// TwinCAT 3 PLC project MAS418_Crane_Simulator_1
// ProgramVersion: 3.1.4024.0
// libraries:
//   Tc2_Standard, * (Beckhoff Automation GmbH)
//   Tc2_System, * (Beckhoff Automation GmbH)
//   Tc3_Module, * (Beckhoff Automation GmbH)
// project tree:
//   Crane_Controller/Enums/ E_ControlBoxSwitchMode.TcDUT, E_RunningStates.TcDUT
//   Crane_Controller/GVL/ G_HMI.TcGVL
//   Crane_Controller/Interfaces/ I_CraneControlBox.TcIO
//   Crane_Controller/POU/ FB_AutoMode.TcPOU, FB_ClosedLoopControl.TcPOU, FB_ControlBox.TcPOU, FB_ManualMode.TcPOU, FB_MotionReferenceGenerator.TcPOU, FB_OpenLoopControl.TcPOU, FB_RealControlBox.TcPOU, FB_VirtualControlBox.TcPOU
//   Crane_Controller/Structs/ ST_CraneHMIData.TcDUT, ST_MotionGeneratorData.TcDUT, ST_OpenLoopControlData.TcDUT
//   / GlobalTextList.TcGTLO, PlcTask.TcTTO, Simulator_1.TcTTO, Visualization Manager.TcVMO (not stored)
//   POUs/ FB_CraneSimulator.TcPOU, MAIN.TcPOU, P_Simulator.TcPOU
//   Task1/ E_SensorBrands.TcDUT, G_Task1.TcGVL, P_Task1.TcPOU
//   Task2/ E_CraneStates.TcDUT, F_DegToRad.TcPOU, F_UpdateParameter.TcPOU, F_UpdateParameterRef.TcPOU, G_Task2.TcGVL, P_Task2.TcPOU, ST_MotorParameters.TcDUT, ST_Timer.TcDUT
//   VISUs/ CraneController.TcVIS, Visualization.TcVIS
// real-time tasks:
//   TASK PlcTask: cycle T#10ms, priority 8, ADS port 350
//   TASK Simulator: cycle T#100us, priority 4, ADS port 351

CONFIGURATION MAS418_Crane_Simulator_1
    RESOURCE PLC ON TwinCAT3
        TASK PlcTask(INTERVAL := T#10ms, PRIORITY := 8);
        TASK Simulator_1(INTERVAL := T#100us, PRIORITY := 4);
        PROGRAM MAIN WITH PlcTask : MAIN;
        PROGRAM P_Simulator WITH Simulator_1 : P_Simulator;
    END_RESOURCE
END_CONFIGURATION

// ---- Crane_Controller/Enums/E_ControlBoxSwitchMode.TcDUT
{attribute 'qualified_only'}
{attribute 'strict'}
TYPE E_ControlBoxSwitchMode :
(
	Off,
	Auto,
	Manual
);
END_TYPE

// ---- Crane_Controller/Enums/E_RunningStates.TcDUT
{attribute 'qualified_only'}
{attribute 'strict'}
TYPE E_RunningStates :
(
	Off,
	Auto,
	Manual
);
END_TYPE

// ---- Crane_Controller/Structs/ST_CraneHMIData.TcDUT
TYPE ST_CraneHMIData :
STRUCT
	eMode				: E_ControlBoxSwitchMode := E_ControlBoxSwitchMode.Off;
	eRunningState 		: E_RunningStates;
	bStart				: BOOL;
	//bStop				: BOOL;
	bAuto				: BOOL;
	bOn					: BOOL;
	//bManual				: BOOL;
	fJoyX				: REAL := 1.6384E+04;
	fJoyY				: REAL := 1.6384e+04;	
	sStatus				: STRING;
END_STRUCT
END_TYPE

// ---- Crane_Controller/Structs/ST_MotionGeneratorData.TcDUT
TYPE ST_MotionGeneratorData :
STRUCT
	fStartPosition_m: LREAL;
	fStartVelocity_m: LREAL;
	fPositionSetpoint_m: LREAL;
	fVelocitySetpoint_m: LREAL;
	fTimeBeforeStarting_s: LREAL;
	fRampTime_s: LREAL;
	fHoldPositionTime_s: LREAL;
END_STRUCT
END_TYPE

// ---- Crane_Controller/Structs/ST_OpenLoopControlData.TcDUT
TYPE ST_OpenLoopControlData :
STRUCT
END_STRUCT
END_TYPE

// ---- Task1/E_SensorBrands.TcDUT
{attribute 'qualified_only'}
{attribute 'strict'}
TYPE E_SensorBrands :
(
	Sick 	:= 0,
	Pilz 	:= 1,
	Parker 	:= 2,
	Bosch 	:= 3
);
END_TYPE

// ---- Task2/E_CraneStates.TcDUT
{attribute 'qualified_only'}
{attribute 'strict'}
TYPE E_CraneStates :
(
	Auto,
	Manual,
	Off
);
END_TYPE

// ---- Task2/ST_MotorParameters.TcDUT
// Task 3
TYPE ST_MotorParameters :
STRUCT
	fMaxSpeed		: REAL;
	fMinSpeed		: REAL;
END_STRUCT
END_TYPE

// ---- Task2/ST_Timer.TcDUT
// Task 2
TYPE ST_Timer :
STRUCT
	bStartTimer				: BOOL				:= FALSE;
	bTimerOutput			: BOOL				:= FALSE;
	tElapsedTime			: TIME				:= T#0S;
	tTimer					: TIME;
END_STRUCT
END_TYPE

// ---- Crane_Controller/GVL/G_HMI.TcGVL
{attribute 'qualified_only'}
VAR_GLOBAL
stHMIVaribles		: ST_CraneHMIData;
END_VAR

// ---- Task1/G_Task1.TcGVL
{attribute 'qualified_only'}
VAR_GLOBAL
	dtCurrentDateTime 		: DATE_AND_TIME;
	tdTimeVar				: TIME 				:= T#5S;
	aArrayOfFourDataTimeVar	: ARRAY[0..3] OF DATE_AND_TIME
	:= [DT#2023-02-07-0:0:10, DT#2023-02-08-0:0:10, DT#2023-02-09-0:0:10, DT#2023-02-10-0:0:10];
	sensor1					: E_SensorBrands 	:= E_SensorBrands.Bosch;
	bStartTimer				: BOOL				:= FALSE;
	bTimerOutput			: BOOL				:= FALSE;
	tElapsedTime			: TIME				:= T#0S;
END_VAR

// ---- Task2/G_Task2.TcGVL
{attribute 'qualified_only'}
VAR_GLOBAL
	// Task 2
	stTimer2			: ST_Timer 	:= (tTimer := T#5S);
	fAngleMotor1Deg		: REAL		:= 180.0;
	fAngleMotor1Rad		: REAL;
	
	// Task 3
	stMotorParameters 	: ST_MotorParameters;
	stMotorParameters2 	: ST_MotorParameters;
END_VAR

// ---- Crane_Controller/Interfaces/I_CraneControlBox.TcIO
INTERFACE I_CraneControlBox
 //   METHOD Mode : E_Mode
 //   METHOD Status : E_RunningStates; 
 //   METHOD Joystick : REAL;

METHOD Joystick : REAL
VAR_INPUT
END_VAR
END_METHOD

METHOD Mode : E_ControlBoxSwitchMode
VAR_INPUT
END_VAR
END_METHOD

METHOD Status : E_RunningStates
VAR_INPUT
END_VAR
END_METHOD

END_INTERFACE

// ---- POUs/MAIN.TcPOU
PROGRAM MAIN
VAR
	//fbVirtualControlBox			: FB_VirtualControlBox;
	
END_VAR

P_Task1();
P_Task2();

END_PROGRAM

// ---- Task1/P_Task1.TcPOU
PROGRAM P_Task1
VAR
	bTestVar 			: BOOL 	:= FALSE;	
	bTestVar2 			: BOOL  := FALSE;
	pDateTime 			: POINTER TO DATE_AND_TIME;
	rTimeVar			: REFERENCE TO TIME := G_Task1.tdTimeVar;
	aInstanceOfArrayOfFourDataTimeVar : ARRAY[0..3] OF DATE_AND_TIME 
	:= G_Task1.aArrayOfFourDataTimeVar;
	fbTon				: TON	:= (PT:=T#10S);
END_VAR

pDateTime := ADR(G_Task1.dtCurrentDateTime);

IF NOT bTestVar THEN
	pDateTime^ := DT#2015-02-04-07:31:19;
	bTestVar := TRUE;
END_IF

IF bTestVar2 THEN
	pDateTime^ := DT#2023-02-08-15:31:19;
	rTimeVar := T#10S;
	aInstanceOfArrayOfFourDataTimeVar[3] := DT#2023-02-25-0:0:10;
	G_Task1.sensor1 := E_SensorBrands.Parker;
END_IF

fbTon(IN := G_Task1.bStartTimer,
	  Q => G_Task1.bTimerOutput,
	  ET => G_Task1.tElapsedTime);

END_PROGRAM

// ---- Task2/P_Task2.TcPOU
PROGRAM P_Task2
VAR
	// Task 2
	fbTof				: TOF	:= (PT:=G_Task2.stTimer2.tTimer);
	
	// Task 3	
	fbRTrig 			: R_TRIG;
	bTriggerd			: BOOL;
	bUpdateMotorSpeed 	: BOOL;
    fNewMotorSpeed 		: REAL := 55.55;
	eCraneStates		: E_CraneStates := E_CraneStates.Off;
	sTestString			: STRING(20);
END_VAR

// Task 2
fbTof(IN := G_Task2.stTimer2.bStartTimer,
	  Q => G_Task2.stTimer2.bTimerOutput,
	  ET => G_Task2.stTimer2.tElapsedTime);

	  
F_DegToRad(fAngleDeg := G_Task2.fAngleMotor1Deg,
		   fAngleRad => G_Task2.fAngleMotor1Rad);
		   
// Task 3
fbRTrig(CLK := bUpdateMotorSpeed,
		Q => bTriggerd);

F_UpdateParameter(bUpdateValue := bTriggerd,
				  fNewValue := fNewMotorSpeed,
				  stMotorParameters := G_Task2.stMotorParameters);
			
F_UpdateParameterRef(bUpdateValue := bTriggerd,
					fNewValue := fNewMotorSpeed,
					stMotorParameters := G_Task2.stMotorParameters2);				  

CASE eCraneStates OF
	E_CraneStates.Off:
		sTestString := 'OFF';
		IF bTriggerd THEN
			eCraneStates := E_CraneStates.Manual;
		END_IF
	E_CraneStates.Manual:
		sTestString := 'Manual';
	E_CraneStates.Auto:
		sTestString := 'Auto';
END_CASE

END_PROGRAM

// ---- Task2/F_DegToRad.TcPOU
// Task 2
FUNCTION F_DegToRad : REAL
VAR_INPUT
	fAngleDeg		: REAL;
END_VAR
VAR
	fPi				: REAL	:= 3.14159265358979323846;
END_VAR
VAR_OUTPUT
	fAngleRad		: REAL;
END_VAR

fAngleRad := fAngleDeg * (fPi/180.0);

END_FUNCTION

// ---- Task2/F_UpdateParameter.TcPOU
FUNCTION F_UpdateParameter : REAL
VAR_INPUT
    bUpdateValue : BOOL;
   	fNewValue : REAL;
	stMotorParameters : ST_MotorParameters;
END_VAR
VAR
END_VAR

	IF bUpdateValue THEN
        stMotorParameters.fMaxSpeed := fNewValue;
    ELSE
        stMotorParameters.fMaxSpeed := stMotorParameters.fMaxSpeed;
    END_IF

END_FUNCTION

// ---- Task2/F_UpdateParameterRef.TcPOU
FUNCTION F_UpdateParameterRef : REAL
VAR_INPUT
    bUpdateValue : BOOL;
   	fNewValue : REAL;
	stMotorParameters : REFERENCE TO ST_MotorParameters;
END_VAR
VAR
END_VAR

	IF bUpdateValue THEN
        stMotorParameters.fMaxSpeed := fNewValue;
    ELSE
        stMotorParameters.fMaxSpeed := stMotorParameters.fMaxSpeed;
    END_IF

END_FUNCTION

// ---- POUs/P_Simulator.TcPOU
PROGRAM P_Simulator
VAR
	fbSimulator 			: FB_CraneSimulator;
	bSimulatorOn 			: BOOL;
	fCylPos 				: LREAL;
	fUDCV					: LREAL;
	ppbar					: LREAL;
	prbar					: LREAL;
	
	
	fbControlboxInterface	: I_CraneControlBox;
	fbVirtualControlbox		: FB_VirtualControlBox;
	
	fbManualMode			: FB_ManualMode;
	fbAutoMode				: FB_AutoMode;
	
	stMotionGeneratorData	: ST_MotionGeneratorData;
END_VAR

//stCraneHMIData REF= G_HMI.stHMIVaribles;

fbControlboxInterface := fbVirtualControlbox;
fbManualMode(fbControlBoxInterface := fbControlboxInterface);
fbAutoMode(fbControlBoxInterface := fbControlboxInterface);

IF fbControlboxInterface.Mode() = E_ControlBoxSwitchMode.Manual THEN
	fbManualMode();
	fUDCV := TO_LREAL(fbManualMode.fUCV);
	
ELSIF fbControlboxInterface.Mode() = E_ControlBoxSwitchMode.Auto THEN
	// Generate data for motion ref
	stMotionGeneratorData.fHoldPositionTime_s := 1.0;
	stMotionGeneratorData.fPositionSetpoint_m := 0.2;
	stMotionGeneratorData.fRampTime_s := 2.0;
	stMotionGeneratorData.fStartPosition_m := fbSimulator.xm;
	stMotionGeneratorData.fStartVelocity_m := 0.0;
	stMotionGeneratorData.fTimeBeforeStarting_s := 2.0;
	stMotionGeneratorData.fVelocitySetpoint_m := 0.02;
	
	fbAutoMode(fbControlBoxInterface := fbControlboxInterface,
			   bEnable := NOT (fbControlboxInterface.Mode() = E_ControlBoxSwitchMode.Off),
			   stMotionGeneratorData := stMotionGeneratorData);
	fUDCV := TO_LREAL(fbAutoMode.fUDCV);
END_IF




fbSimulator(
	ssMethodType 	:= BOOL_TO_SINT(NOT (fbControlboxInterface.Mode() = E_ControlBoxSwitchMode.Off)),
	uDCV			:= fUDCV,
	xm 				=> fCylPos,
	ppbar 			=> ppbar,
	prbar			=> prbar);

END_PROGRAM

// ---- POUs/FB_CraneSimulator.TcPOU
FUNCTION_BLOCK FB_CraneSimulator
VAR_INPUT
	ssMethodType: SINT;
	uDCV: LREAL;
END_VAR
VAR_OUTPUT
	xm: LREAL;
	ppbar: LREAL;
	prbar: LREAL;
END_VAR
VAR
	pLS: LREAL;
	QDCV_out: LREAL;
	rtb_xDot: LREAL;
	rtb_xDotDot: LREAL;
	temp1: LREAL;
	temp2: LREAL;
	temp3: LREAL;
	temp4: LREAL;
	c_DiscreteTimeIntegrator2_D: LREAL;
	c_DiscreteTimeIntegrator3_D: LREAL;
	c_DiscreteTimeIntegrator_DS: LREAL;
	c_DiscreteTimeIntegrator4_D: LREAL;
END_VAR



CASE ssMethodType OF
    0: //SS_INITIALIZE: 
        (* SystemInitialize for Atomic SubSystem: '<Root>/FB_CraneSimulator' *)
        (* InitializeConditions for DiscreteIntegrator: '<S1>/Discrete-Time Integrator' *)
        c_DiscreteTimeIntegrator_DS := 4.377E+6;
        (* InitializeConditions for DiscreteIntegrator: '<S1>/Discrete-Time Integrator2' *)
        c_DiscreteTimeIntegrator2_D := 0.0;
        (* InitializeConditions for DiscreteIntegrator: '<S1>/Discrete-Time Integrator3' *)
        c_DiscreteTimeIntegrator3_D := 0.0;
        (* InitializeConditions for DiscreteIntegrator: '<S1>/Discrete-Time Integrator4' *)
        c_DiscreteTimeIntegrator4_D := 468300.0;
        (* End of SystemInitialize for SubSystem: '<Root>/FB_CraneSimulator' *)
    1: //SS_STEP: 
        (* Outputs for Atomic SubSystem: '<Root>/FB_CraneSimulator' *)
        (* DiscreteIntegrator: '<S1>/Discrete-Time Integrator2' *)
        rtb_xDot := c_DiscreteTimeIntegrator2_D;
        (* Outport: '<Root>/x [m]' incorporates:
         *  DiscreteIntegrator: '<S1>/Discrete-Time Integrator3' *)
        xm := c_DiscreteTimeIntegrator3_D;
        (* Outport: '<Root>/pp [bar]' incorporates:
         *  DiscreteIntegrator: '<S1>/Discrete-Time Integrator'
         *  Gain: '<S1>/Gain' *)
        ppbar := 1.0E-5 * c_DiscreteTimeIntegrator_DS;
        (* Outport: '<Root>/pr [bar]' incorporates:
         *  DiscreteIntegrator: '<S1>/Discrete-Time Integrator4'
         *  Gain: '<S1>/Gain1' *)
        prbar := 1.0E-5 * c_DiscreteTimeIntegrator4_D;
        (* MATLAB Function: '<S1>/MATLAB Function' incorporates:
         *  DiscreteIntegrator: '<S1>/Discrete-Time Integrator'
         *  DiscreteIntegrator: '<S1>/Discrete-Time Integrator2'
         *  DiscreteIntegrator: '<S1>/Discrete-Time Integrator3'
         *  DiscreteIntegrator: '<S1>/Discrete-Time Integrator4' *)
        (* Parameters *)
        (* MATLAB Function 'FB_CraneSimulator/MATLAB Function': '<S2>:1' *)
        (* '<S2>:1:3' Fexternal = 1.3365e+04; *)
        (* [N] *)
        (* '<S2>:1:4' mEffective = 1.3365e+04; *)
        (* [kg] *)
        (* '<S2>:1:5' kFric = 4000; *)
        (* [N/(ms)] *)
        (* '<S2>:1:6' Apiston = 0.0033; *)
        (* [m^2] *)
        (* '<S2>:1:7' Aannulus = 0.0023; *)
        (* [m^2] *)
        (* '<S2>:1:8' beta = 1.0e9; *)
        (* [Pa] *)
        (* '<S2>:1:9' pSupply = 180e5; *)
        (* [Pa] *)
        (* '<S2>:1:10' pReturn = 1.1e5; *)
        (* [Pa] *)
        (* '<S2>:1:11' MaxStroke = 0.5; *)
        (* [m] *)
        (* '<S2>:1:12' VCyl_A = 1.0e-03; *)
        (* '<S2>:1:13' VCyl_B = 1.25e-03; *)
        (* '<S2>:1:14' p_nom_DCV = 7e5; *)
        (* '<S2>:1:15' Q1_ref_DCV = 20/6e4; *)
        (* '<S2>:1:16' kv1_DCV = Q1_ref_DCV/sqrt(p_nom_DCV); *)
        (* '<S2>:1:17' p0 = 7e5; *)
        (* compensator crack pressure *)
        (* Directional Control Valve - Lifting Cylinder  *)
        (* LS Pressure *)
        (* '<S2>:1:20' if uDCV > 0 *)

        IF uDCV > 0.0 THEN 
            (* '<S2>:1:21' pLS = pPiston; *)
            pLS := c_DiscreteTimeIntegrator_DS;
        ELSIF uDCV < 0.0 THEN 
            (* '<S2>:1:22' elseif uDCV < 0 *)
            (* '<S2>:1:23' pLS = pRod; *)
            pLS := c_DiscreteTimeIntegrator4_D;
        ELSE 
            (* '<S2>:1:24' else *)
            (* '<S2>:1:25' pLS = 0; *)
            pLS := 0.0;
        END_IF;

        (* '<S2>:1:28' if pLS<0 *)

        IF pLS < 0.0 THEN 
            (* '<S2>:1:29' pLS = 0; *)
            pLS := 0.0;
        END_IF;

        (* Pressure Compensator *)
        (* '<S2>:1:33' pPC = 0; *)
        (* '<S2>:1:35' if p0 <= (pSupply - pLS) *)

        IF (1.8E+7 - pLS) >= 700000.0 THEN 
            (* '<S2>:1:36' pPC = pLS+p0; *)
            pLS := pLS + 700000.0;
        ELSE 
            (* '<S2>:1:37' elseif 0 < (pSupply - pLS) < p0 *)
            (* '<S2>:1:38' pPC = pSupply-pLS; *)
            pLS := 1.8E+7 - pLS;
        END_IF;

        (* '<S2>:1:43' if pPC<0 *)

        IF pLS < 0.0 THEN 
            (* '<S2>:1:44' pPC = 0; *)
            pLS := 0.0;
        END_IF;

        (* Orifice Equations *)
        (* '<S2>:1:47' if uDCV > 0 *)

        IF uDCV > 0.0 THEN 
            (* '<S2>:1:48' QDCV_in =  kv1_DCV*uDCV*sign(pPC-pPiston)*sqrt(abs(pPC-pPiston)); *)
            pLS := pLS - c_DiscreteTimeIntegrator_DS;

            IF pLS < 0.0 THEN 
                rtb_xDotDot := -1.0;
            ELSIF pLS > 0.0 THEN 
                rtb_xDotDot := 1.0;
            ELSE 
                rtb_xDotDot := 0.0;
            END_IF;

            temp3 := ABS(pLS);
            pLS := ((3.9840953644479785E-7 * uDCV) * rtb_xDotDot) * SQRT(temp3);
            (* '<S2>:1:49' QDCV_out = kv1_DCV*uDCV*sign(pRod-pReturn)*sqrt(abs(pRod-pReturn)); *)

            IF (c_DiscreteTimeIntegrator4_D - 110000.0) < 0.0 THEN 
                rtb_xDotDot := -1.0;
            ELSIF (c_DiscreteTimeIntegrator4_D - 110000.0) > 0.0 THEN 
                rtb_xDotDot := 1.0;
            ELSE 
                rtb_xDotDot := 0.0;
            END_IF;

            temp4 := ABS(c_DiscreteTimeIntegrator4_D - 110000.0);
            QDCV_out := ((3.9840953644479785E-7 * uDCV) * rtb_xDotDot) * SQRT(temp4);
        ELSIF uDCV < 0.0 THEN 
            (* '<S2>:1:50' elseif uDCV < 0 *)
            (* '<S2>:1:51' QDCV_out =  kv1_DCV*uDCV*sign(pPC-pRod)*sqrt(abs(pPC-pRod)); *)
            pLS := pLS - c_DiscreteTimeIntegrator4_D;

            IF pLS < 0.0 THEN 
                rtb_xDotDot := -1.0;
            ELSIF pLS > 0.0 THEN 
                rtb_xDotDot := 1.0;
            ELSE 
                rtb_xDotDot := 0.0;
            END_IF;

            temp1 := ABS(pLS);
            QDCV_out := ((3.9840953644479785E-7 * uDCV) * rtb_xDotDot) * SQRT(temp1);
            (* '<S2>:1:52' QDCV_in =  kv1_DCV*uDCV*sign(pRod-pReturn)*sqrt(abs(pRod-pReturn)); *)

            IF (c_DiscreteTimeIntegrator4_D - 110000.0) < 0.0 THEN 
                rtb_xDotDot := -1.0;
            ELSIF (c_DiscreteTimeIntegrator4_D - 110000.0) > 0.0 THEN 
                rtb_xDotDot := 1.0;
            ELSE 
                rtb_xDotDot := 0.0;
            END_IF;

            temp2 := ABS(c_DiscreteTimeIntegrator4_D - 110000.0);
            pLS := ((3.9840953644479785E-7 * uDCV) * rtb_xDotDot) * SQRT(temp2);
        ELSE 
            (* '<S2>:1:53' else *)
            (* '<S2>:1:54' QDCV_in = 0; *)
            pLS := 0.0;
            (* '<S2>:1:55' QDCV_out = 0; *)
            QDCV_out := 0.0;
        END_IF;

        (* Pressure Gradients *)
        (* '<S2>:1:58' VA = VCyl_A + x*Apiston; *)
        (* '<S2>:1:59' VB =  VCyl_B + (MaxStroke - x)*Aannulus; *)
        (* '<S2>:1:60' VA_dot = Apiston*xDot; *)
        (* '<S2>:1:61' VB_dot = -Aannulus*xDot; *)
        (* '<S2>:1:62' pPistonDot = beta/VA*(QDCV_in - VA_dot); *)
        (* '<S2>:1:63' pRodDot = beta/VB*(-QDCV_out - VB_dot); *)
        QDCV_out := (1.0E+9 / (((0.5 - c_DiscreteTimeIntegrator3_D) * 0.0023) + 0.00125)) * (( -QDCV_out) - (-0.0023 * c_DiscreteTimeIntegrator2_D));
        (* Viscouse Friction *)
        (* '<S2>:1:66' Ffric = kFric*xDot; *)
        (* Hydraulic Force *)
        (* '<S2>:1:69' Fhyd = pPiston*Apiston - pRod*Aannulus; *)
        (* Newton Second Law of Motion *)
        (* '<S2>:1:72' xDotDot = (Fhyd - Ffric - Fexternal)/mEffective; *)
        rtb_xDotDot := ((((c_DiscreteTimeIntegrator_DS * 0.0033) - (c_DiscreteTimeIntegrator4_D * 0.0023)) - (4000.0 * c_DiscreteTimeIntegrator2_D)) - 13365.0) / 13365.0;
        (* Update for DiscreteIntegrator: '<S1>/Discrete-Time Integrator' incorporates:
         *  DiscreteIntegrator: '<S1>/Discrete-Time Integrator2'
         *  DiscreteIntegrator: '<S1>/Discrete-Time Integrator3'
         *  MATLAB Function: '<S1>/MATLAB Function' *)
        c_DiscreteTimeIntegrator_DS := (((1.0E+9 / ((c_DiscreteTimeIntegrator3_D * 0.0033) + 0.001)) * (pLS - (0.0033 * c_DiscreteTimeIntegrator2_D))) * 0.0001) + c_DiscreteTimeIntegrator_DS;

        IF c_DiscreteTimeIntegrator_DS >= 1.8E+7 THEN 
            c_DiscreteTimeIntegrator_DS := 1.8E+7;
        ELSIF c_DiscreteTimeIntegrator_DS <= 110000.0 THEN 
            c_DiscreteTimeIntegrator_DS := 110000.0;
        END_IF;

        (* End of Update for DiscreteIntegrator: '<S1>/Discrete-Time Integrator' *)
        

        (* Update for DiscreteIntegrator: '<S1>/Discrete-Time Integrator2' *)
        c_DiscreteTimeIntegrator2_D := (0.0001 * rtb_xDotDot) + c_DiscreteTimeIntegrator2_D;

        IF c_DiscreteTimeIntegrator2_D >= 0.12 THEN 
            c_DiscreteTimeIntegrator2_D := 0.12;
        ELSIF c_DiscreteTimeIntegrator2_D <= -0.12 THEN 
            c_DiscreteTimeIntegrator2_D := -0.12;
        END_IF;

        (* End of Update for DiscreteIntegrator: '<S1>/Discrete-Time Integrator2' *)
        

        (* Update for DiscreteIntegrator: '<S1>/Discrete-Time Integrator3' *)
        c_DiscreteTimeIntegrator3_D := (0.0001 * rtb_xDot) + c_DiscreteTimeIntegrator3_D;

        IF c_DiscreteTimeIntegrator3_D >= 0.5 THEN 
            c_DiscreteTimeIntegrator3_D := 0.5;
        ELSIF c_DiscreteTimeIntegrator3_D <= 0.0 THEN 
            c_DiscreteTimeIntegrator3_D := 0.0;
        END_IF;

        (* End of Update for DiscreteIntegrator: '<S1>/Discrete-Time Integrator3' *)
        

        (* Update for DiscreteIntegrator: '<S1>/Discrete-Time Integrator4' *)
        c_DiscreteTimeIntegrator4_D := (0.0001 * QDCV_out) + c_DiscreteTimeIntegrator4_D;

        IF c_DiscreteTimeIntegrator4_D >= 1.8E+7 THEN 
            c_DiscreteTimeIntegrator4_D := 1.8E+7;
        ELSIF c_DiscreteTimeIntegrator4_D <= 110000.0 THEN 
            c_DiscreteTimeIntegrator4_D := 110000.0;
        END_IF;

        (* End of Update for DiscreteIntegrator: '<S1>/Discrete-Time Integrator4' *)
        (* End of Outputs for SubSystem: '<Root>/FB_CraneSimulator' *)
END_CASE;

END_FUNCTION_BLOCK

// ---- Crane_Controller/POU/FB_VirtualControlBox.TcPOU
FUNCTION_BLOCK FB_VirtualControlBox IMPLEMENTS I_CraneControlBox
VAR_INPUT
		//_stCranHMIVaribels		: REFERENCE TO ST_CraneHMIData;
END_VAR
VAR_OUTPUT
END_VAR
VAR
	_stCranHMIVaribels			: REFERENCE TO ST_CraneHMIData := G_HMI.stHMIVaribles;
END_VAR

METHOD Joystick : REAL;

VAR 
	fTemp		: REAL;
END_VAR
//fTemp := _stCranHMIVaribels.fJoyX * 2.0/32767.0 - 1;

fTemp:= _stCranHMIVaribels.fJoyX * 0.1/32767.0 - 0.05;


IF ABS(fTemp) <= 0.005 THEN
	Joystick := 0.0;
ELSE
	Joystick := fTemp;
END_IF
END_METHOD

METHOD Mode : E_ControlBoxSwitchMode
UpdateRunningMode();
Mode := _stCranHMIVaribels.eMode;
END_METHOD

METHOD OLD_FB_init : BOOL
VAR_INPUT
	bInitRetains : BOOL; // if TRUE, the retain variables are initialized (warm start / cold start)
	bInCopyCode : BOOL;  // if TRUE, the instance afterwards gets moved into the copy code (online change)
	stCranHMIVaribels : REFERENCE TO ST_CraneHMIData;
END_VAR
_stCranHMIVaribels := stCranHMIVaribels;
END_METHOD

METHOD Status : E_RunningStates


VAR 
	eTemp : E_RunningStates;
END_VAR
UpdateRunningMode();

//IF stCranHMIVaribels.eMode = E_ControlBoxSwitchMode.Off AND NOT (stCranHMIVaribels.eRunningState = E_RunningStates.Ready)THEN
//	stCranHMIVaribels.eRunningState := E_RunningStates.NotReady;
//ELSIF (stCranHMIVaribels.eMode = E_ControlBoxSwitchMode.Manual) OR (stCranHMIVaribels.eMode = E_ControlBoxSwitchMode.Auto) THEN
//	stCranHMIVaribels.eRunningState := E_RunningStates.Ready;
//ELSIF stCranHMIVaribels.bStart THEN
//	stCranHMIVaribels.eRunningState := E_RunningStates.Starting;
//ELSIF (stCranHMIVaribels.eRunningState = E_RunningStates.Ready) THEN
//	stCranHMIVaribels.eRunningState := E_RunningStates.Running;
//ELSIF (stCranHMIVaribels.eMode = E_ControlBoxSwitchMode.Off) AND (Joystick() <= 0.01) THEN
//	stCranHMIVaribels.eRunningState := E_RunningStates.Stopping;
//END_IF

//Status := stCranHMIVaribels.eRunningState;



IF Mode() = E_ControlBoxSwitchMode.Off THEN
	eTemp := E_RunningStates.NotReady;
	_stCranHMIVaribels.eRunningState := eTemp;
	Status := eTemp;
	RETURN;
ELSIF NOT (Mode() = E_ControlBoxSwitchMode.Off) AND NOT (_stCranHMIVaribels.eRunningState = E_RunningStates.Running) THEN
	eTemp := E_RunningStates.Ready;	
END_IF

IF _stCranHMIVaribels.bStart AND NOT (_stCranHMIVaribels.eRunningState = E_RunningStates.Running) THEN
	eTemp := E_RunningStates.Starting;
END_IF

IF NOT (Mode() = E_ControlBoxSwitchMode.Off) AND _stCranHMIVaribels.bStart THEN
	eTemp := E_RunningStates.Running;
END_IF

IF NOT _stCranHMIVaribels.bStart AND ABS(Joystick()) >= 0.01 THEN
	eTemp := E_RunningStates.Stopping;
END_IF

_stCranHMIVaribels.sStatus := TO_STRING(eTemp);
_stCranHMIVaribels.eRunningState := eTemp;
Status := eTemp;
END_METHOD

METHOD PRIVATE UpdateRunningMode : REAL
VAR_INPUT
END_VAR
VAR
END_VAR
IF NOT _stCranHMIVaribels.bOn THEN
	_stCranHMIVaribels.eMode := E_ControlBoxSwitchMode.Off;
	RETURN;
ELSIF _stCranHMIVaribels.bAuto THEN
	_stCranHMIVaribels.eMode := E_ControlBoxSwitchMode.Manual;
ELSE
	_stCranHMIVaribels.eMode := E_ControlBoxSwitchMode.Auto; 
END_IF
END_METHOD

END_FUNCTION_BLOCK

// ---- Crane_Controller/POU/FB_ManualMode.TcPOU
FUNCTION_BLOCK FB_ManualMode
VAR_INPUT
	fbControlBoxInterface			: REFERENCE TO I_CraneControlBox;
END_VAR
VAR_OUTPUT
	fUCV					: REAL;
	bEnable					: BOOL;
END_VAR
VAR
	//fbVirtualControlbox		: FB_VirtualControlBox;
	//fbControlBox			: I_CraneControlBox := fbVirtualControlbox;
	fbOpenLoopController 	: FB_OpenLoopControl;
	fVelRefFromJoy			: REAL;
END_VAR

fVelRefFromJoy := fbControlBoxInterface.Joystick();

IF NOT(fbControlBoxInterface.Mode() = E_ControlBoxSwitchMode.Off) THEN
	bEnable := TRUE;
ELSE
	bEnable := FALSE;	
END_IF

fbOpenLoopController(bEnable := bEnable,
					 fVRef := fVelRefFromJoy);

fUCV := fbOpenLoopController.fUDCV;

END_FUNCTION_BLOCK

// ---- Crane_Controller/POU/FB_OpenLoopControl.TcPOU
FUNCTION_BLOCK FB_OpenLoopControl
VAR_INPUT
	bEnable			: BOOL;
	fVRef			: REAL;

END_VAR
VAR_OUTPUT
	fUDCV			: REAL;
END_VAR
VAR
	fTemp			: REAL;
	fBoreArea		: REAL := 0.0033183;
	fAnnulusArea	: REAL := 0.0023562;
	fQMax			: REAL := 20.0;
END_VAR

IF bEnable THEN
	
	IF fVRef <= 0 THEN
		fTemp := fVRef*fBoreArea*60000.0;
	ELSE
		fTemp := fVRef*fAnnulusArea*60000.0;
	END_IF
	
fUDCV := fTemp/fQMax;
ELSE
	fUDCV := 0;
END_IF

END_FUNCTION_BLOCK

// ---- Crane_Controller/POU/FB_AutoMode.TcPOU
FUNCTION_BLOCK FB_AutoMode
VAR_INPUT
	fbControlBoxInterface		: REFERENCE TO I_CraneControlBox;
	stMotionGeneratorData		: ST_MotionGeneratorData;
	bEnable						: BOOL;
END_VAR
VAR_OUTPUT
	fUDCV 						: REAL;
END_VAR
VAR
	fbColsedLoopController		: FB_ClosedLoopControl;
	fbOpenLoopController		: FB_OpenLoopControl;
	fbMotionGen					: FB_MotionReferenceGenerator;
	fbTon						: TON;
END_VAR

IF NOT (fbControlBoxInterface.Mode() = E_ControlBoxSwitchMode.Off) THEN
	fUDCV := 0;
	RETURN;
END_IF

// Start timer
fbTon(IN := bEnable,
	  PT := T#100000MS);

fbMotionGen(bEnable 	:= bEnable,
			fClock_s	:= TO_REAL(fbTon.ET),
			fStartPosition_m := stMotionGeneratorData.fStartPosition_m,
			fStartVelocity_m := stMotionGeneratorData.fStartVelocity_m,
			fPositionSetpoint_m := stMotionGeneratorData.fPositionSetpoint_m,
			fVelocitySetpoint_m := stMotionGeneratorData.fVelocitySetpoint_m,
			fTimeBeforeStarting_s := stMotionGeneratorData.fTimeBeforeStarting_s,
			fRampTime_s := stMotionGeneratorData.fRampTime_s,
			fHoldPositionTime_s := stMotionGeneratorData.fHoldPositionTime_s);
			
fbOpenLoopController(bEnable := bEnable,
					fVRef := fbMotionGen.fVelocityReference_m);

fbColsedLoopController(bEnable := bEnable,
						fPositionRef := fbMotionGen.fPositionReference_m);
						
fUDCV := fbColsedLoopController.fUPFB + fbOpenLoopController.fUDCV;

END_FUNCTION_BLOCK

// ---- Crane_Controller/POU/FB_ClosedLoopControl.TcPOU
FUNCTION_BLOCK FB_ClosedLoopControl
VAR_INPUT
	bEnable				: BOOL;
	fPGain				: REAL;
	fPositionRef		: REAL;
	fPositionFeedback	: REAL;
END_VAR
VAR_OUTPUT
	fPositionError		: REAL;
	fUPFB				: REAL;
END_VAR
VAR
END_VAR

IF bEnable THEN
	fUPFB := (fPositionRef - fPositionFeedback)*fPGain;

ELSE
	fUPFB := 0.0;
END_IF

END_FUNCTION_BLOCK

// ---- Crane_Controller/POU/FB_MotionReferenceGenerator.TcPOU
FUNCTION_BLOCK FB_MotionReferenceGenerator
VAR_INPUT
	bEnable: BOOL;
	fStartPosition_m: LREAL;
	fStartVelocity_m: LREAL;
	fPositionSetpoint_m: LREAL;
	fVelocitySetpoint_m: LREAL;
	fTimeBeforeStarting_s: LREAL;
	fRampTime_s: LREAL;
	fHoldPositionTime_s: LREAL;
	fClock_s: LREAL;
END_VAR
VAR_OUTPUT
	fPositionReference_m: LREAL;
	fVelocityReference_m: LREAL;
	fTotalMotionTime_s: LREAL;
	fErrorSignal: LREAL;
END_VAR
VAR
	Error: DINT;
	slopeExt: LREAL;
	tHold: LREAL;
	x1: LREAL;
	x4: LREAL;
	rtb_Saturation3: LREAL;
	x1_tmp: LREAL;
	x1_tmp_tmp: LREAL;
	x4_tmp: LREAL;
	x4_tmp_tmp: LREAL;
	x4_tmp_tmp_0: LREAL;
	x4_tmp_tmp_1: LREAL;
	x1_tmp_0: LREAL;
END_VAR


(* Outputs for Atomic SubSystem: '<Root>/FB_MotionReferenceGenerator' *)
(* Saturate: '<S1>/Saturation2' *)

IF fVelocitySetpoint_m > 0.05 THEN 
    fPositionReference_m := 0.05;
ELSIF fVelocitySetpoint_m >= 0.0 THEN 
    fPositionReference_m := fVelocitySetpoint_m;
ELSE 
    fPositionReference_m := 0.0;
END_IF;

(* End of Saturate: '<S1>/Saturation2' *)


(* Saturate: '<S1>/Saturation3' *)

IF fPositionSetpoint_m > 0.45 THEN 
    rtb_Saturation3 := 0.45;
ELSIF fPositionSetpoint_m >= 0.0 THEN 
    rtb_Saturation3 := fPositionSetpoint_m;
ELSE 
    rtb_Saturation3 := 0.0;
END_IF;

(* End of Saturate: '<S1>/Saturation3' *)


(* MATLAB Function: '<S1>/WaveSignal' *)
(* MATLAB Function 'FB_MotionReferenceGenerator/WaveSignal': '<S2>:1' *)
(* '<S2>:1:2' x_SP = x_ref - x0; *)
(* '<S2>:1:3' vs=v_ref; *)
(* '<S2>:1:4' slopeExt=v0-vs; *)
slopeExt := fStartVelocity_m - fPositionReference_m;
(* '<S2>:1:5' slopeRetr=-vs-v0; *)
(* '<S2>:1:7' as = vs/tRamp; *)
(* '<S2>:1:8' s_acc=(vs^2-v0^2)/as; *)
(* '<S2>:1:10' tHold=(x_SP-s_acc)/vs; *)
tHold := ((rtb_Saturation3 - fStartPosition_m) - (((fPositionReference_m * fPositionReference_m) - (fStartVelocity_m * fStartVelocity_m)) / (fPositionReference_m / fRampTime_s))) / fPositionReference_m;
(* '<S2>:1:12' if tHold < 0 *)

IF tHold < 0.0 THEN 
    (* '<S2>:1:13' Error = 1; *)
    Error := 1;
ELSE 
    (* '<S2>:1:14' else *)
    (* '<S2>:1:15' Error = 0; *)
    Error := 0;
END_IF;

(* '<S2>:1:18' t1=tRamp; *)
(* '<S2>:1:19' t2=tHold; *)
(* '<S2>:1:20' t3=tRamp; *)
(* '<S2>:1:21' t4=tWait; *)
(* '<S2>:1:22' t5=t1; *)
(* '<S2>:1:23' t6=t2; *)
(* '<S2>:1:24' t7=t3; *)
(* '<S2>:1:26' x = x0; *)
(* '<S2>:1:27' x1 = x0 + v0*((t0+t1)-t0)-(slopeExt/t1)*((t0+t1)-t0)^2/2; *)
x1_tmp_tmp := fTimeBeforeStarting_s + fRampTime_s;
x1_tmp := x1_tmp_tmp - fTimeBeforeStarting_s;
x1_tmp_0 := slopeExt / fRampTime_s;
x1 := ((x1_tmp * fStartVelocity_m) + fStartPosition_m) - ((x1_tmp_0 * (x1_tmp * x1_tmp)) / 2.0);
(* '<S2>:1:28' x2 = x1 + vs*((t0+t1+t2)-(t0+t1)); *)
(* '<S2>:1:29' x4 = x_ref - v0*((t0+t1+t2+t3+t4+t5)-(t0+t1+t2+t3+t4))+(slopeRetr/t5)*((t0+t1+t2+t3+t4+t5)-(t0+t1+t2+t3+t4))^2/2; *)
x4_tmp_tmp := x1_tmp_tmp + tHold;
x4_tmp_tmp_0 := x4_tmp_tmp + fRampTime_s;
x4_tmp := x4_tmp_tmp_0 + fHoldPositionTime_s;
x4_tmp_tmp_1 := x4_tmp + fRampTime_s;
x4 := x4_tmp_tmp_1 - x4_tmp;
x1_tmp := (( -fPositionReference_m) - fStartVelocity_m) / fRampTime_s;
x4 := (rtb_Saturation3 - (x4 * fStartVelocity_m)) + ((x1_tmp * (x4 * x4)) / 2.0);
(* '<S2>:1:30' x5 = x4-vs*((t0+t1+t2+t3+t4+t5+t6)-(t0+t1+t2+t3+t4+t5)); *)
(* '<S2>:1:32' if Error == 1 *)

IF Error = 1 THEN 
    (* '<S2>:1:33' x = x0; *)
    rtb_Saturation3 := fStartPosition_m;
    (* '<S2>:1:34' v = v0; *)
    fPositionReference_m := fStartVelocity_m;
ELSIF (fClock_s >= 0.0) AND (fClock_s < fTimeBeforeStarting_s) THEN 
    (* '<S2>:1:35' elseif t>=0 && t<t0 *)
    (* '<S2>:1:36' x = x0; *)
    rtb_Saturation3 := fStartPosition_m;
    (* '<S2>:1:37' v = v0; *)
    fPositionReference_m := fStartVelocity_m;
ELSIF (fClock_s >= fTimeBeforeStarting_s) AND (fClock_s < x1_tmp_tmp) THEN 
    (* '<S2>:1:38' elseif t>=t0 && t<(t0+t1) *)
    (* '<S2>:1:39' x = x0 + v0*(t-t0)-(slopeExt/t1)*(t-t0)^2/2; *)
    x4_tmp_tmp_0 := fClock_s - fTimeBeforeStarting_s;
    rtb_Saturation3 := ((x4_tmp_tmp_0 * fStartVelocity_m) + fStartPosition_m) - ((x1_tmp_0 * (x4_tmp_tmp_0 * x4_tmp_tmp_0)) / 2.0);
    (* '<S2>:1:40' v = v0-(slopeExt/t1)*(t-t0); *)
    fPositionReference_m := fStartVelocity_m - (x1_tmp_0 * x4_tmp_tmp_0);
ELSIF (fClock_s >= x1_tmp_tmp) AND (fClock_s < x4_tmp_tmp) THEN 
    (* '<S2>:1:41' elseif t>=(t0+t1) && t<(t0+t1+t2) *)
    (* '<S2>:1:42' x = x1 + vs*(t-(t0+t1)); *)
    rtb_Saturation3 := ((fClock_s - x1_tmp_tmp) * fPositionReference_m) + x1;
    (* '<S2>:1:43' v = vs; *)
ELSIF (fClock_s >= x4_tmp_tmp) AND (fClock_s < x4_tmp_tmp_0) THEN 
    (* '<S2>:1:44' elseif t>=(t0+t1+t2) && t<(t0+t1+t2+t3) *)
    (* '<S2>:1:45' x = x2+vs*(t-(t0+t1+t2))+(slopeExt/t3)*(t-(t0+t1+t2))^2/2; *)
    x4_tmp_tmp_0 := fClock_s - x4_tmp_tmp;
    rtb_Saturation3 := ((((x4_tmp_tmp - x1_tmp_tmp) * fPositionReference_m) + x1) + (x4_tmp_tmp_0 * fPositionReference_m)) + ((x1_tmp_0 * (x4_tmp_tmp_0 * x4_tmp_tmp_0)) / 2.0);
    (* '<S2>:1:46' v = vs+(slopeExt/t3)*(t-(t0+t1+t2)); *)
    fPositionReference_m := (x4_tmp_tmp_0 * (slopeExt / fRampTime_s)) + fPositionReference_m;
ELSIF (fClock_s >= x4_tmp_tmp_0) AND (fClock_s < x4_tmp) THEN 
    (* '<S2>:1:47' elseif t>=(t0+t1+t2+t3) && t<(t0+t1+t2+t3+t4) *)
    (* '<S2>:1:48' x = x_ref; *)
    (* '<S2>:1:49' v = v0; *)
    fPositionReference_m := fStartVelocity_m;
ELSIF (fClock_s >= x4_tmp) AND (fClock_s < x4_tmp_tmp_1) THEN 
    (* '<S2>:1:50' elseif t>=(t0+t1+t2+t3+t4) && t<(t0+t1+t2+t3+t4+t5) *)
    (* '<S2>:1:51' x = x_ref - v0*(t-(t0+t1+t2+t3+t4))+(slopeRetr/t5)*(t-(t0+t1+t2+t3+t4))^2/2; *)
    slopeExt := fClock_s - x4_tmp;
    rtb_Saturation3 := (rtb_Saturation3 - (slopeExt * fStartVelocity_m)) + ((x1_tmp * (slopeExt * slopeExt)) / 2.0);
    (* '<S2>:1:52' v = v0+(slopeRetr/t5)*(t-(t0+t1+t2+t3+t4)); *)
    fPositionReference_m := (slopeExt * x1_tmp) + fStartVelocity_m;
ELSE 
    rtb_Saturation3 := x4_tmp_tmp_1 + tHold;

    IF (fClock_s >= x4_tmp_tmp_1) AND (fClock_s < rtb_Saturation3) THEN 
        (* '<S2>:1:53' elseif t>=(t0+t1+t2+t3+t4+t5) && t<(t0+t1+t2+t3+t4+t5+t6) *)
        (* '<S2>:1:54' x = x4-vs*(t-(t0+t1+t2+t3+t4+t5)); *)
        rtb_Saturation3 := x4 - ((fClock_s - x4_tmp_tmp_1) * fPositionReference_m);
        (* '<S2>:1:55' v = -vs; *)
        fPositionReference_m :=  -fPositionReference_m;
    ELSIF (fClock_s >= rtb_Saturation3) AND (fClock_s < (rtb_Saturation3 + fRampTime_s)) THEN 
        (* '<S2>:1:56' elseif t>=(t0+t1+t2+t3+t4+t5+t6) && t<(t0+t1+t2+t3+t4+t5+t6+t7) *)
        (* '<S2>:1:57' x = x5-vs*(t-(t0+t1+t2+t3+t4+t5+t6))-(slopeRetr/t3)*(t-(t0+t1+t2+t3+t4+t5+t6))^2/2; *)
        x4_tmp_tmp_0 := fClock_s - rtb_Saturation3;
        rtb_Saturation3 := ((x4 - ((rtb_Saturation3 - x4_tmp_tmp_1) * fPositionReference_m)) - (x4_tmp_tmp_0 * fPositionReference_m)) - ((x1_tmp * (x4_tmp_tmp_0 * x4_tmp_tmp_0)) / 2.0);
        (* '<S2>:1:58' v = -vs-(slopeRetr/t3)*(t-(t0+t1+t2+t3+t4+t5+t6)); *)
        fPositionReference_m := ( -fPositionReference_m) - (x4_tmp_tmp_0 * x1_tmp);
    ELSE 
        (* '<S2>:1:59' else *)
        (* '<S2>:1:60' x = x0; *)
        rtb_Saturation3 := fStartPosition_m;
        (* '<S2>:1:61' v = v0; *)
        fPositionReference_m := fStartVelocity_m;
    END_IF;

END_IF;

(* Switch: '<S1>/Switch' *)
(* '<S2>:1:64' T = t0+t1+t2+t3+t4+t5+t6+t7; *)

IF  NOT bEnable THEN 
    fPositionReference_m := fStartVelocity_m;
END_IF;

(* End of Switch: '<S1>/Switch' *)


(* Saturate: '<S1>/Saturation' *)

IF fPositionReference_m > 0.05 THEN 
    (* Outport: '<Root>/fVelocityReference_m' *)
    fVelocityReference_m := 0.05;
ELSIF fPositionReference_m >= -0.05 THEN 
    (* Outport: '<Root>/fVelocityReference_m' *)
    fVelocityReference_m := fPositionReference_m;
ELSE 
    (* Outport: '<Root>/fVelocityReference_m' *)
    fVelocityReference_m := -0.05;
END_IF;

(* End of Saturate: '<S1>/Saturation' *)


(* Switch: '<S1>/Switch1' *)

IF bEnable THEN 
    fPositionReference_m := rtb_Saturation3;
ELSE 
    fPositionReference_m := fStartPosition_m;
END_IF;

(* End of Switch: '<S1>/Switch1' *)


(* Saturate: '<S1>/Saturation1' *)

IF fPositionReference_m > 0.45 THEN 
    (* Outport: '<Root>/fPositionReference_m' *)
    fPositionReference_m := 0.45;
ELSIF fPositionReference_m < 0.0 THEN 
    (* Outport: '<Root>/fPositionReference_m' *)
    fPositionReference_m := 0.0;
END_IF;

(* End of Saturate: '<S1>/Saturation1' *)


(* Outport: '<Root>/fTotalMotionTime_s' incorporates:
 *  MATLAB Function: '<S1>/WaveSignal' *)
fTotalMotionTime_s := ((((((fTimeBeforeStarting_s + fRampTime_s) + tHold) + fRampTime_s) + fHoldPositionTime_s) + fRampTime_s) + tHold) + fRampTime_s;
(* Outport: '<Root>/fErrorSignal' incorporates:
 *  MATLAB Function: '<S1>/WaveSignal' *)
fErrorSignal := DINT_TO_LREAL(Error);
(* End of Outputs for SubSystem: '<Root>/FB_MotionReferenceGenerator' *)

END_FUNCTION_BLOCK

// ---- Crane_Controller/POU/FB_ControlBox.TcPOU
FUNCTION_BLOCK FB_ControlBox
VAR_INPUT
END_VAR
VAR_OUTPUT
END_VAR
VAR
	_iControlBox	: REFERENCE TO I_CraneControlBox;
END_VAR

METHOD FB_init : BOOL
VAR_INPUT
	bInitRetains : BOOL; // if TRUE, the retain variables are initialized (warm start / cold start)
	bInCopyCode : BOOL;  // if TRUE, the instance afterwards gets moved into the copy code (online change)
	iControlBox		: REFERENCE TO I_CraneControlBox;
END_VAR
_iControlBox := iControlBox;
END_METHOD

METHOD Joystick : REAL
VAR_INPUT
END_VAR
Joystick := _iControlBox.Joystick();
END_METHOD

END_FUNCTION_BLOCK

// ---- Crane_Controller/POU/FB_RealControlBox.TcPOU
FUNCTION_BLOCK FB_RealControlBox IMPLEMENTS I_CraneControlBox
VAR_INPUT
END_VAR
VAR_OUTPUT
END_VAR
VAR
END_VAR

{warning 'add method implementation '}
METHOD Joystick : REAL
Joystick := 0.0;
END_METHOD

{warning 'add method implementation '}
METHOD Mode : E_ControlBoxSwitchMode
Mode := E_ControlBoxSwitchMode.Off;
END_METHOD

{warning 'add method implementation '}
METHOD Status : E_RunningStates
Status := E_RunningStates.NotReady;
END_METHOD

END_FUNCTION_BLOCK

// ---- GlobalTextList.TcGTLO
TEXTLIST GlobalTextList
  984 = '%f'
  306 = '%s'
  981 = 'Auto'
  837 = 'Crane Controller'
  757 = 'Crane Simulator'
  439 = 'dd'
  609 = 'Joy_X'
  265 = 'Joy_Y'
  597 = 'Manual'
  939 = 'Mode'
  276 = 'Off'
  696 = 'On/Off'
  706 = 'Position [m]'
  373 = 'pp'
  504 = 'pr'
  154 = 'Start'
  415 = 'Status'
  258 = 'Stop'
  809 = 'uDCV'
END_TEXTLIST

// ---- VISUs/CraneController.TcVIS
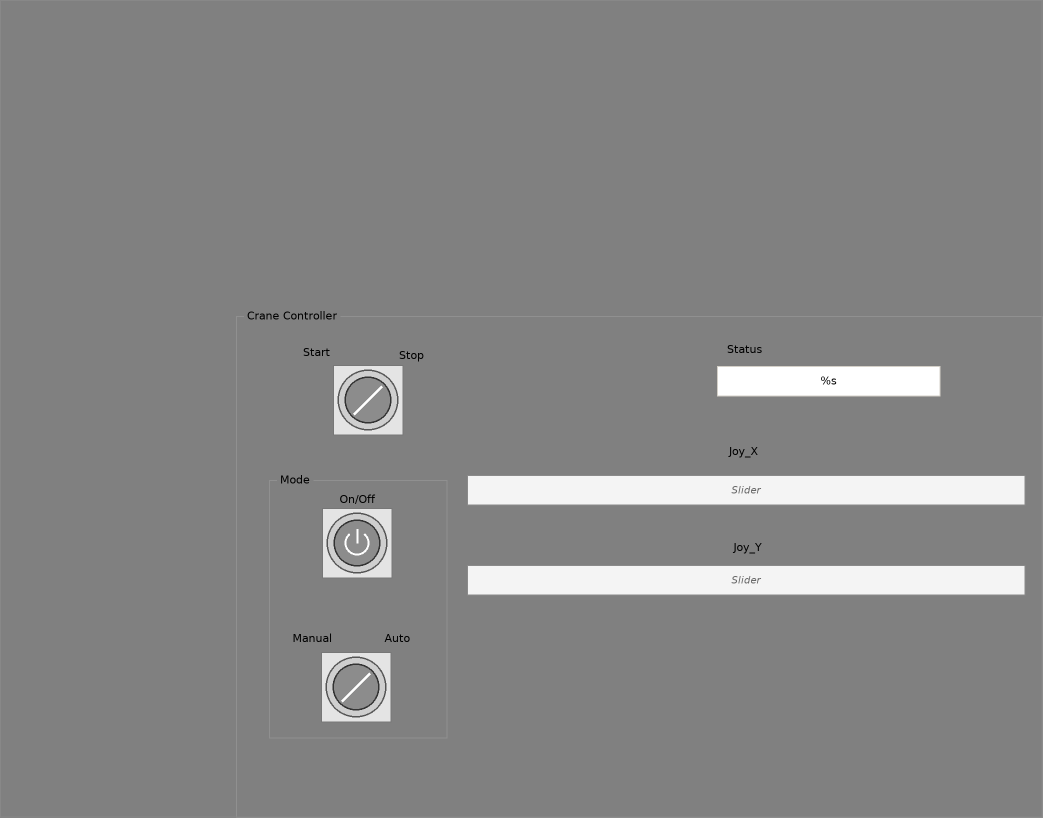
VISUALIZATION CraneController  // 1043x818
    GroupBox (236,308 807x510), "Crane Controller"
        GroupBox (33,164 178x266), "Mode"
            Label (61,14 55x27), "On/Off"
            Label (101,153 55x27), "Auto"
            PowerSwitch (53,36 70x70), variable: G_HMI.stHMIVaribles.bOn, behaviour: TOGGLE, style: Switch-PowerSwitch-Gray
            RotarySwitch (52,180 70x70), variable: G_HMI.stHMIVaribles.bAuto, behaviour: TOGGLE, style: Switch-RotarySwitch-Gray
            Label (16,153 55x27), "Manual"
        Textfield (481,58 223x30), "%s", text variable: G_HMI.stHMIVaribles.sStatus
        Label (484,226 55x27), "Joy_Y"
        Label (480,130 55x27), "Joy_X"
        Slider (231,257 558x30), variable: G_HMI.stHMIVaribles.fJoyY, scale 0..100
        Label (481,28 55x27), "Status"
        RotarySwitch (97,57 70x70), variable: G_HMI.stHMIVaribles.bStart, behaviour: TOGGLE, style: Switch-RotarySwitch-Gray
        Label (53,31 55x27), "Start"
        Label (148,34 55x27), "Stop"
        Slider (231,167 558x30), variable: G_HMI.stHMIVaribles.fJoyX, scale 0..32767
END_VISUALIZATION

// ---- VISUs/Visualization.TcVIS
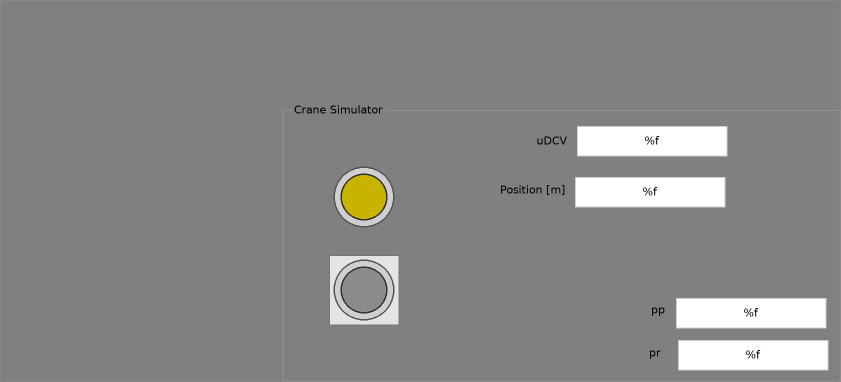
VISUALIZATION Visualization  // 841x382
    GroupBox (283,102 558x280), "Crane Simulator"
        Lamp1 (46,60 70x70), variable: G_HMI.stHMIVaribles.bOn, style: Lamp-Lamp1-Yellow
        PushSwitch (46,153 70x70), variable: P_Simulator.bSimulatorOn, behaviour: TOGGLE, style: Switch-PushSwitch-Gray
        Textfield (294,24 150x30), "%f", text variable: P_Simulator.fUDCV
        Textfield (292,75 150x30), "%f", text variable: P_Simulator.fCylPos
        Textfield (393,196 150x30), "%f", text variable: P_Simulator.ppbar
        Textfield (395,238 150x30), "%f", text variable: P_Simulator.prbar
        Label (194,24 150x30), "uDCV"
        Label (175,73 150x30), "Position [m]"
        Label (300,193 150x30), "pp"
        Label (297,236 150x30), "pr"
END_VISUALIZATION
